(* PLC project 117_1_V0.5.project, CODESYS CODESYS V3.5 SP17 Patch 3 *)
(* stored: creationDateTime 1970-01-01T00:00:00, modificationDateTime 2026-06-16T22:51:19.9979415 *)

FUNCTION_BLOCK SM3ServoDriver
  VAR_INPUT
    TimeManager : REFERENCE TO TimeManager;
  END_VAR
  VAR
    _CheckAxisCommuniction : SMC_CheckAxisCommunication;  (* Проверка связи с драйвером *)
    _CheckPowerStatus : MC_ReadBoolParameter;  (* Прверка питания драйвера *)
    _pNum : UINT;
    _powerStatusValue : ARRAY[0..1] OF BOOL;
    _Power : MC_Power;  (* Управление питанием драйвера *)
    _powerSteps : UINT;
    _Jogging : MC_Jog;  (* Ручной режим *)
    _FollowVelocity : SMC_FollowVelocity;  (* Режим управления скоростью *)
    _Reset_Errors : MC_Reset;  (* Сброс аварий *)
    _reset_Enable : BOOL;
    _bErrors : ARRAY[communication..(lastIndex - 1)] OF BOOL;  (* Дата и время для логов Сбор ошобок в слово *)
    _wAxisErrors : BYTE;
    _ErrorsFlag : BOOL;
    _eAxisErrorsID : ARRAY[communication..(lastIndex - 1)] OF SMC_ERROR;  (* Данные для флагов ошибок и записи в лог *)
    _sComments : ARRAY[communication..(lastIndex - 1)] OF STRING(40);
    _trErrorsTrigs : ARRAY[communication..(lastIndex - 1)] OF R_TRIG;
    _axisErrorsLog : ARRAY[0..9] OF STRING(100);  (* Лог *)
    _logSize : UINT;
    _errorIndex : ERROR_INDEX;
  END_VAR
  VAR CONSTANT
    dPowerParameter : ARRAY[0..1] OF DINT := [1015, 1016];
  END_VAR

            // Проверка связи
_CheckAxisCommuniction(
	Axis	:= SM_Drive_GenericDSP402,
	bEnable := TRUE);

//Проверка наличия питания
FOR _pNum := 0 TO 1 DO
	_CheckPowerStatus(
		Axis			:= SM_Drive_GenericDSP402,
		Enable			:= TRUE,
		ParameterNumber	:= dPowerParameter[_pNum],
		Value			=> _powerStatusValue[_pNum]); 
END_FOR

// Питание драйвера
_Power(Axis	:= SM_Drive_GenericDSP402);

// Ручное управление дравером
_Jogging(Axis := SM_Drive_GenericDSP402); 

//Режим управления скоростью
_FollowVelocity(Axis := SM_Drive_GenericDSP402);

// Сброс ошибок
_Reset_Errors(Axis:= SM_Drive_GenericDSP402, Execute:= _reset_Enable); 

// // Запись флагов ошибок ФБ в массив
// _bErrors[communication]	 := _CheckAxisCommuniction.bError;
// _bErrors[power]			 := _Power.Error;
// _bErrors[jogging]		 := _Jogging.Error;
// _bErrors[follow]		 := _FollowVelocity.bError;
// _bErrors[reset]			 := _Reset_Errors.Error;

// Запись ошибок
FOR _errorIndex := communication TO lastIndex - 1 DO
	// Триггеры ошибок для записи в лог	
	_trErrorsTrigs[_errorIndex](CLK := _bErrors[_errorIndex]);
	
	// 	Формирование слова ошибок
    IF _bErrors[_errorIndex] THEN
        _wAxisErrors := _wAxisErrors OR SHL(BYTE#1, _errorIndex);
	ELSE
		_wAxisErrors := _wAxisErrors AND NOT SHL(BYTE#1, _errorIndex);
    END_IF
	
END_FOR

// Идентификаторы ошибок
_eAxisErrorsID	[communication]	:= _CheckAxisCommuniction.eErrorID;
_eAxisErrorsID	[power]			:= _Power.ErrorID;
_eAxisErrorsID	[jogging]		:= _Jogging.ErrorID;
_eAxisErrorsID	[follow]		:= _FollowVelocity.iErrorID;
_eAxisErrorsID	[reset]			:= _Reset_Errors.ErrorID;

//Коментарии к ошибкам
_sComments		[communication] := 'Ошибка при диагностике связи';
_sComments		[power]			:= 'Ошибка при включении питания драйвера';
_sComments		[jogging]		:= 'Ошибка при ручном управлении';
_sComments		[follow]		:= 'Ошибка при управлении скоростью';
_sComments		[reset]			:= 'Ошибка при сбросе ошибок';

// Метод для записи ошибки в лог
FOR _errorIndex := communication TO lastIndex - 1 DO
_error_handler(
	bError		:= _trErrorsTrigs[_errorIndex].Q,
	arrIndex	:= _errorIndex,
	eErrorID	:= _eAxisErrorsID[_errorIndex],
	sComment	:= _sComments[_errorIndex]
);	
END_FOR

_ErrorsFlag	:= _wAxisErrors > 0;





          

METHOD set_power_on : BOOL
  VAR_INPUT
    powerState : BOOL := FALSE;
  END_VAR
                  

CASE _powerSteps OF
	0:
		IF powerState THEN
			set_power_on := _Power.Status;
		ELSE
			_powerSteps	:= _powerSteps + 1;	
		END_IF
		
	1: 
		_Power.Enable		:= TRUE;
		_Power.bRegulatorOn := TRUE;
		_Power.bDriveStart	:= TRUE;
		_powerSteps			:= _powerSteps + 1;
	2:
		IF _Power.Status THEN 
			_Power.Enable	:= FALSE;
			_powerSteps		:= _powerSteps + 1;
		END_IF
	3: 
			_Power.bRegulatorOn := FALSE;
			_Power.bDriveStart	:= FALSE;
			set_power_on		:= TRUE;
			_powerSteps			:= 0;
END_CASE

                
END_METHOD

METHOD stop_follow_velocity : BOOL
                  _FollowVelocity.bExecute		:= FALSE;
_FollowVelocity.fSetVelocity	:= 0.0; 
	
stop_follow_velocity := _FollowVelocity.bBusy; 
                
END_METHOD

METHOD start_forward_jogging : BOOL
  VAR_INPUT
    velocity : LREAL := 0;
    acceleration : LREAL := 0;
    deceleration : LREAL := 0;
    jerk : LREAL := 0;
  END_VAR
                  _Jogging.JogForward		:= TRUE; 
_Jogging.JogBackward	:= FALSE; 
_Jogging.Velocity		:= velocity; 
_Jogging.Acceleration	:= acceleration; 
_Jogging.Deceleration	:= deceleration; 
_Jogging.Jerk			:= jerk; 

start_forward_jogging := _Jogging.Busy;
                
END_METHOD

(* Проверка питания драйвера *)
METHOD get_power_status : BOOL
                  get_power_status := _powerStatusValue[0] AND _powerStatusValue[1] AND _Power.Status AND _Power.Status;



                
END_METHOD

METHOD set_power_off : BOOL
  VAR_INPUT
    powerState : BOOL;
  END_VAR
                  IF powerState THEN
	set_power_off := TRUE;
	RETURN;
ELSE
	CASE _powerSteps OF
		0: 
			_Power.Enable		:= TRUE;
			_Power.bRegulatorOn := FALSE;
			_Power.bDriveStart	:= FALSE;
			_powerSteps			:= _powerSteps + 1;
		1:
			_Power.Enable	:= FALSE;
			_powerSteps			:= _powerSteps + 1;
		2:
			IF NOT _Power.Status THEN
				set_power_off	:= TRUE;
				_powerSteps		:= 0;
			END_IF
	END_CASE
END_IF

                
END_METHOD

METHOD stop_jogging : BOOL
  VAR_INPUT
    velocity : LREAL := 0;
    acceleration : LREAL := 0;
    deceleration : LREAL := 0;
    jerk : LREAL := 0;
  END_VAR
                  _Jogging.JogForward		:= FALSE; 
_Jogging.JogBackward	:= FALSE; 
_Jogging.Velocity		:= 0; 
_Jogging.Acceleration	:= 0; 
_Jogging.Deceleration	:= 0; 
_Jogging.Jerk			:= 0; 

stop_jogging := _Jogging.Busy;
                
END_METHOD

METHOD reset_errors : BOOL
                  _reset_Enable := TRUE;
IF _Reset_Errors.Done THEN
	reset_errors := _Reset_Errors.Done;
	_reset_Enable := FALSE;
END_IF
                
END_METHOD

METHOD start_follow_velocity : BOOL
  VAR_INPUT
    velocity : LREAL := 0;
  END_VAR
                  _FollowVelocity.bExecute		:= TRUE;
_FollowVelocity.fSetVelocity	:= velocity; 
	
start_follow_velocity := _FollowVelocity.bBusy; 

                
END_METHOD

METHOD get_axis_errors : BOOL
  VAR_INPUT
    errorIndex : ERROR_INDEX;
  END_VAR
                  

get_axis_errors := _bErrors[errorIndex];
                
END_METHOD

METHOD start_backward_jogging : BOOL
  VAR_INPUT
    velocity : LREAL := 0;
    acceleration : LREAL := 0;
    deceleration : LREAL := 0;
    jerk : LREAL := 0;
  END_VAR
                  _Jogging.JogForward		:= FALSE; 
_Jogging.JogBackward	:= TRUE; 
_Jogging.Velocity		:= velocity; 
_Jogging.Acceleration	:= acceleration; 
_Jogging.Deceleration	:= deceleration; 
_Jogging.Jerk			:= jerk; 

start_backward_jogging := _Jogging.Busy;
                
END_METHOD

METHOD _error_handler : BOOL
  VAR_INPUT
    bError : BOOL;
    arrIndex : ERROR_INDEX;
    eErrorID : SMC_ERROR;
    sComment : STRING;
  END_VAR
  VAR
    sDT : STRING;
    toStringError : SMC_ERROR_TO_STRING;
  END_VAR
                  // Запускаем блок даты и времени
IF bError THEN
// Приводим дату и время к типу STRING
	sDT := (DT_TO_STRING(TimeManager.get_date_time()));
// Проиводим SMC_ERROR к перечислению которое умеет в TO_STRING
	toStringError := TO_WORD(eErrorID);
// Cобираем сообщение	
	_axisErrorsLog[_logSize] := CONCAT(RIGHT(sDT,LEN(sDT)-3),': ');
	_axisErrorsLog[_logSize] := CONCAT(_axisErrorsLog[_logSize], TO_STRING(toStringError));
	_axisErrorsLog[_logSize] := CONCAT(_axisErrorsLog[_logSize],' ,');
	_axisErrorsLog[_logSize] := CONCAT(_axisErrorsLog[_logSize],sComment);
// Двигаем индекс массива	
	IF _logSize >= 9 THEN
		_logSize := 0;
	ELSE	
		_logSize := _logSize + 1;
	END_IF	
END_IF

                
END_METHOD

(* Поверка связи с дравером *)
METHOD get_axis_communication : BOOL
                  get_axis_communication := _CheckAxisCommuniction.bOperational;


                
END_METHOD
END_FUNCTION_BLOCK
